// TIA Portal V17 export
// export: Created 2023-04-03T06:31:43.6404026Z, ExportSetting WithDefaults, DisplayName Totally Integrated Automation Portal, DisplayVersion V17 Update 4, DisplayName TIA Portal Openness, DisplayVersion V17 Update 4, DisplayName TIA Portal Version Control Interface, DisplayVersion V17, DisplayName STEP 7 Professional, DisplayVersion V17 Update 4, DisplayName STEP 7 Safety, DisplayVersion V17, DisplayName WinCC Professional, DisplayVersion V17 Update 4
TYPE "PCS"
// stored: IsFailsafeCompliant false
   STRUCT
      iAssetSt : Int;
      rPac : Real;
      rSac : Real;
      rQac : Real;
      iCodeSt : Int;
      rIdcBus1 : Real;
      rPdcBus1 : Real;
      rVdcBus1 : Real;
      DriveSt : Int;
      FreqRef : Real;
      rFreq : Real;
      Mref : Real;
      Nref : Real;
      OperMode : Int;
      rPacBus1Ref : Real;
      rQacBus1Ref : Real;
      rIr : Real;
      rVrs : Real;
      rIs : Real;
      rVst : Real;
      rIt : Real;
      rVtr : Real;
      Vref : Real;
      rIdcBus2 : Real;
      rPdcBus2 : Real;
      rVdcBus2 : Real;
      rPacBus2Ref : Real;
      rQacBus2Ref : Real;
   END_STRUCT;
END_TYPE
